SUBAPPLICATION Uebung_010bA2 (* Toggle Flip-Flop mit IE AuxFunction2_X1 AuxEnabled *)
  (* Standard: 61499-2; Description: Copyright (c) 2023 Meisterschulen am Ostbahnhof This program and the accompanying materials are made available under the terms of the Eclipse Public License 2.0 which is available at https://www.eclipse.org/legal/epl-2.0/ SPDX-License-Identifier: EPL-2.0 *)
  (* Version 1.0, 2023-10-23, Franz Höpfinger, Meisterschulen am Ostbahnhof, initial API and implementation and/or initial documentation *)
  PACKAGE Uebungen;
  IMPORT Uebungen::const::UT::DefaultPool::AuxFunction2_X1;
  IMPORT isobus::UT::io::Auxiliary::IN::AuxiliaryState;
  IMPORT logiBUS::io::DQ::logiBUS_DO::Output_Q1;
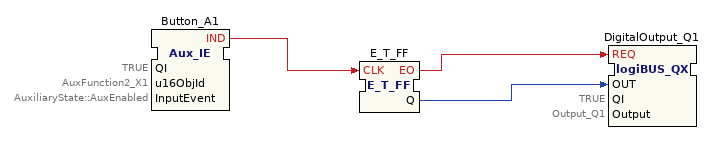
  (* AuxEnabled wird nicht wiederholt bei einem AUX Type 2 bei Aux Type 0 schon. Lange drücken ergibt 1 Event bei Type 2 Bool_Latched = 0,    /**< Two-position switch */ Bool_NonLatched = 2,    /**< Two-position switch - returns to off */ *)
  FBS
    DigitalOutput_Q1 : logiBUS::io::DQ::logiBUS_QX(QI := TRUE, Output := Output_Q1);
    Button_A1 : isobus::UT::io::Auxiliary::IN::Aux_IE(QI := TRUE, u16ObjId := AuxFunction2_X1, InputEvent := AuxiliaryState::AuxEnabled);
    E_T_FF : iec61499::events::E_T_FF;
  END_FBS
  EVENT_CONNECTIONS
    Button_A1.IND TO E_T_FF.CLK;
    E_T_FF.EO TO DigitalOutput_Q1.REQ;
  END_CONNECTIONS
  DATA_CONNECTIONS
    E_T_FF.Q TO DigitalOutput_Q1.OUT;
  END_CONNECTIONS
END_SUBAPPLICATION
